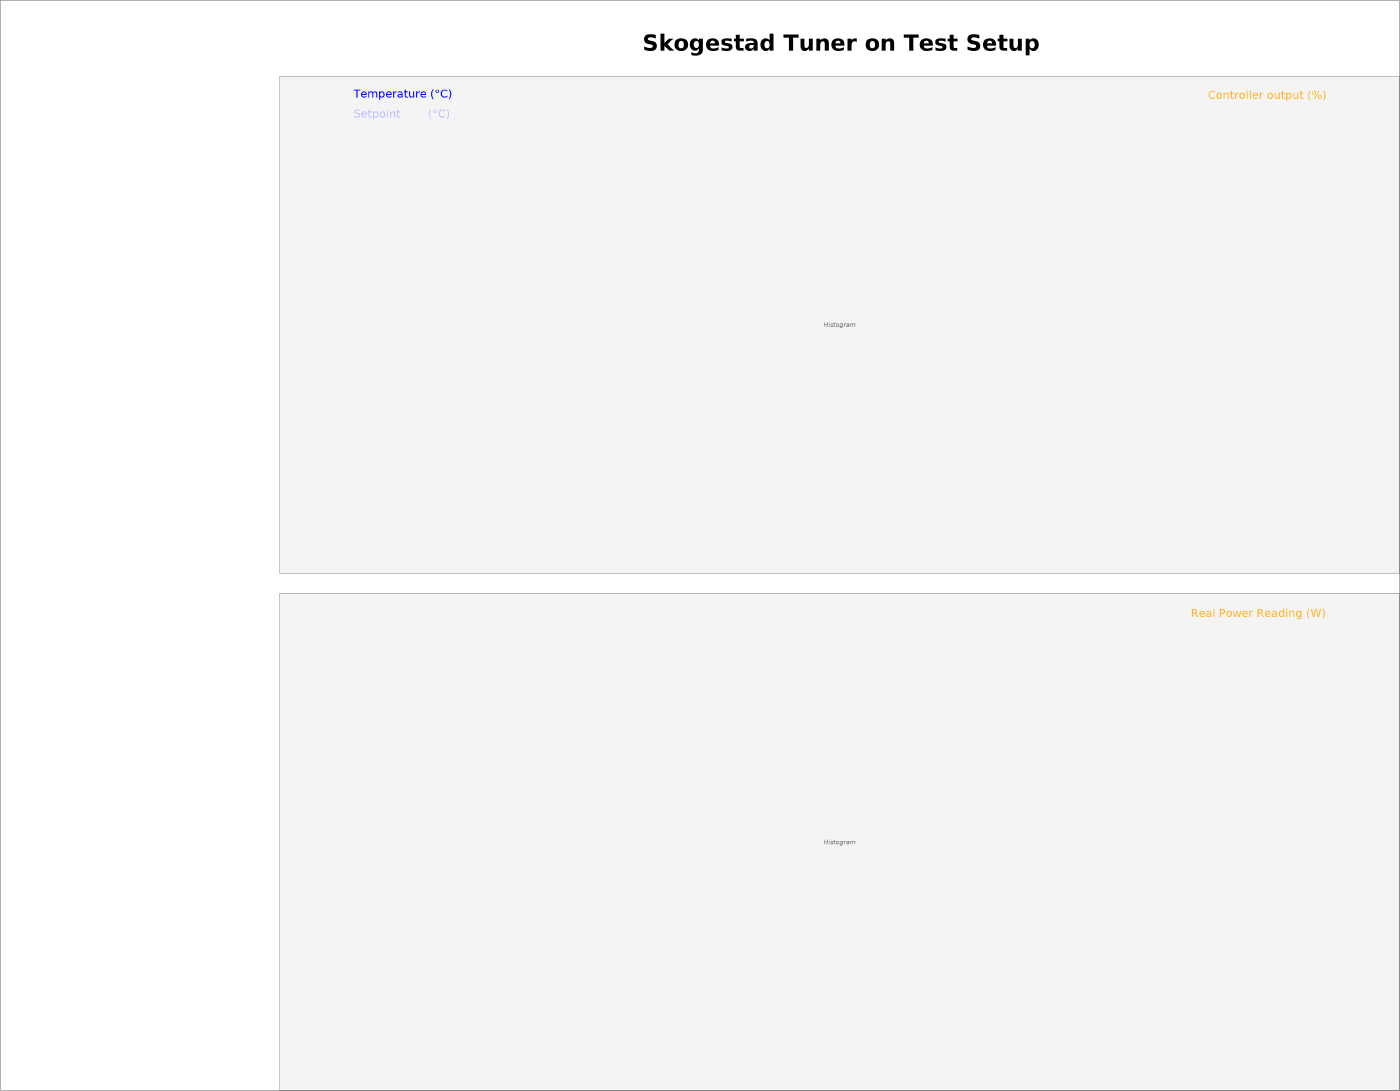
VISUALIZATION Visualization  // 2249x1754
    Histogram (449,122 1800x800), scale format: %.1f, scale 0..100
        p1518820177: GVL.arTempData
        p102497268: GVL.arTempData
        p788070771: ARRAY [0..2000] OF REAL
    Histogram (449,122 1800x800), scale format: %.1f, scale 0..100
        p1518820177: GVL.arControllerData
        p102497268: GVL.arControllerData
        p788070771: ARRAY [0..2000] OF INT
    Histogram (449,122 1800x800), scale format: %.1f, scale 0..100
        p1518820177: GVL.arSetpointData
        p102497268: GVL.arSetpointData
        p788070771: ARRAY [0..20000] OF REAL
    Label (565,136 167x30), "Temperature (°C)"
    Label (1941,138 193x30), "Controller output (%)"
    Label (1022,36 659x66), "Skogestad Tuner on Test Setup"
    Histogram (449,954 1800x800), scale format: %.1f, scale 0..160
        p1518820177: GVL.arRealPowerData
        p102497268: GVL.arRealPowerData
        p788070771: ARRAY [0..10000] OF INT
    Label (1901,971 232x30), "Real Power Reading (W)"
    Label (565,168 167x30), "Setpoint (°C)"
END_VISUALIZATION

(* stored: Version 1.1.0.1, ProductVersion 3.1.4024.12
   Visu Visualization: Id {f5eb54d4-7d38-4be2-9a4e-22252c25c95e} *)
